// TIA Portal V18 export
TYPE "LGasp_typeCmdAutoAttuatore"
// stored: IsFailsafeCompliant false
   STRUCT
      startcicloauto : Bool;   // Cmd start --> posizionamento se asse , ciclo stampo se EV
      autopos : Bool;   // Cmd jog positivo
      autoneg : Bool;   // Cmd jog negativo
   END_STRUCT;
END_TYPE
